Staubli VAL3: start.pgx

program start()
begin
  //
  call Init()
  call Main()


end
